PROGRAM Q2
VAR
END_VAR

(*
SFC, Sequential Function Chart
Operations are represented with states that have transition conditions.
Operations are run whilst the containing state is active.

Advantages include:
	Easy to get basic states implemented
	Transition conditions are very clear
	May have operations on the entry or exit of a state
	
Disadvantages include:
	More intricate operations are a bit tricky to implement
	Concurrent operations are more difficult or repetitive to implement

*)

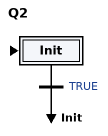
INITIAL_STEP Init:
END_STEP
TRANSITION FROM Init TO Init
    := TRUE;
END_TRANSITION

END_PROGRAM

(* stored: Version 1.1.0.1, ProductVersion 3.1.4024.12
   POU Q2: Id {dd9f9d89-3bc7-4017-9fd0-ecfdcf38c4e4}, SpecialFunc None *)
